Universal Robots PolyScope program: a_full_up.urp

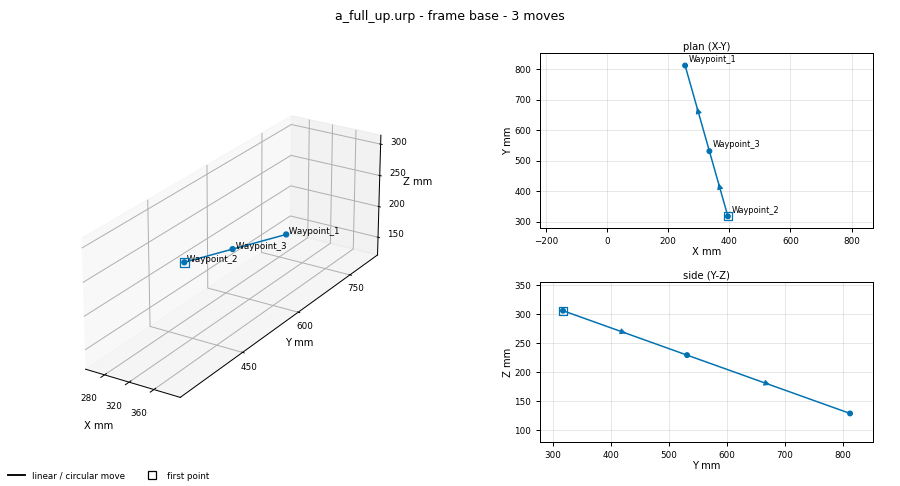
[picture p0: tool path of a_full_up.urp in frame base, 3 of 3 moves have a stored position in this frame; points joined in program order, loops and branches not executed]
Program a_full_up (installation=string_planes directory=/programs createdIn=5.17.3 lastSavedIn=5.17.3 robotSerialNumber=20245501435)
Calibrated DH parameters: a=[0.000154, -0.137004, -0.385524, -0.00002, 0.000092, 0]; d=[0.162441, 211.794786, -230.585024, 18.923638, 0.099786, 0.09951]; alpha=[1.569493, -0.001902, 0.003874, 1.570111, -1.570167, 0]; deltaTheta=[0, -1.242934, 1.056292, 0.186646, 0.000002, 0.000001]
InitVariablesNode
Robot Program (runOnlyOnce=false)
  MoveL speed 250 mm/s, acceleration 1200 mm/s^2 (useActiveTCP=true) feature=Joint_6_name
    Waypoint Waypoint_2: TCP in base x=395.327 y=317.91 z=305.826 mm, rx=1.7389 ry=2.3104 rz=-1.1078 rad; joints [-161.343, -67.838, 103.559, -90.294, -114.046, -169.479] deg; TCP offset x=28.21 y=-96.107 z=-99.69 mm, rx=0 ry=0 rz=0 rad; feature pose in base x=395.332 y=317.908 z=305.826 mm, rx=1.7389 ry=2.3104 rz=-1.1077 rad
    Waypoint Waypoint_3: motionParameters(blendRadius=0.05); TCP in base x=334.761 y=531.331 z=229.441 mm, rx=1.7389 ry=2.3104 rz=-1.1078 rad; joints [-140.937, -50.825, 87.453, -85.938, -101.389, -152.604] deg; feature pose in base x=334.76 y=531.325 z=229.425 mm, rx=1.7389 ry=2.3104 rz=-1.1078 rad
    Waypoint Waypoint_1: TCP in base x=255.207 y=811.658 z=129.108 mm, rx=1.7389 ry=2.3104 rz=-1.1078 rad; joints [-122.369, -14.783, 31.291, -64.48, -89.14, -138.649] deg; feature pose in base x=255.21 y=811.658 z=129.122 mm, rx=1.7389 ry=2.3105 rz=-1.1078 rad
